Fanuc KAREL source: ARRAY_LEN.kl

PROGRAM T
%NOLOCKGROUP
VAR
 v0 : ARRAY[5] OF INTEGER
 res : INTEGER
BEGIN
 res = ARRAY_LEN(v0)
END T
